FUNCTION_BLOCK FB_TIMETRACKER
VAR_INPUT
END_VAR
VAR_OUTPUT
	TimeStamp		: DT;
END_VAR
VAR
	GetSystemTime	: FB_LOCALSYSTEMTIME;
	TimeStampStruct	: TIMESTRUCT;
END_VAR

GetSystemTime(sNetID := '', bEnable := TRUE, systemTime => TimeStampStruct);
TimeStamp := SYSTEMTIME_TO_DT(TimeStampStruct);

END_FUNCTION_BLOCK

(* stored: Version 1.1.0.1, ProductVersion 3.1.4024.12
   POU FB_TIMETRACKER: Id {ee573b6e-a6be-4aea-b740-dd4ae5b155fa}, SpecialFunc None *)
